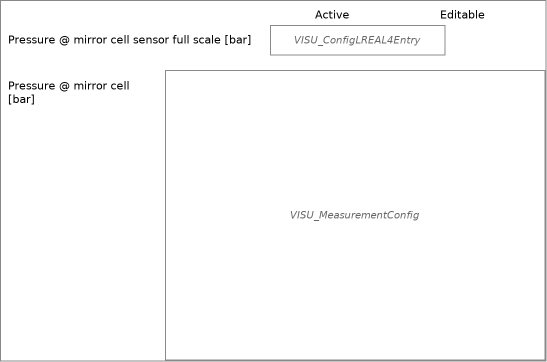
VISUALIZATION VISU_M1Config_Radial_MirrorPressure  // 547x362
VAR_IN_OUT
    editable : M1RadialSupportConfig;
	active : M1RadialSupportConfig;
END_VAR
    Label (270,5 125x20), "Active"
    Label (400,5 125x20), "Editable"
    Label (5,25 260x30), "Pressure @ mirror cell sensor full scale [bar]"
    Frame (270,25 175x30)
        shows VISU_ConfigLREAL4Entry(active := active.mirrorPressureSensorFullScale, editable := editable.mirrorPressureSensorFullScale)
    Label (5,60 145x65), "Pressure @ mirror cell [bar]"
    Frame (165,70 380x290)
        shows VISU_MeasurementConfig(active := active.mirrorPressure, editable := editable.mirrorPressure)
END_VISUALIZATION

(* stored: Version 1.1.0.1, ProductVersion 3.1.4019.2
   Visu VISU_M1Config_Radial_MirrorPressure: Id {a7e3fa10-d227-461c-9d85-6d6225929481} *)
